// TIA Portal V20 export
TYPE "LConSMC_typeUnitConfiguration"
// Konfiguration der Einheiten / Configuration of the units
// stored: Access Published
   STRUCT
      metricUnits : Bool := TRUE;   // TRUE: Verwendung metrischer Einheiten [m] / [m/min] / [m/s^2] / [N] FALSE: Verwendung angloamerikanischer Einheiten [inch] / [ft/min] / [ft/s^2] / [Lbf] / TRUE: Use metric system [m] / [m/min] / [m/s^2] / [N] FALSE: Use angloamerican system [inch] / [ft/min] / [ft/s^2] / [Lbf]
      axisVelocityUnit : UDInt := 1083;   // Geschwindigkeitseinheit des Technologieobjektes (siehe TO.Units.VelocityUnit) !Nur notwendig wenn "getAxisConfigAtStart" = FALSE! / Velocity unit of TO (see TO.Units.VelocityUnit) !Only necessary if "getAxisConfigAtStart" = FALSE!
      axisTorqueUnit : UDInt := 1126;   // Drehmomenteinheit des Technologieobjektes (siehe TO.Units.TorqueUnit) !Nur notwendig wenn "getAxisConfigAtStart" = FALSE! / Torque unit of TO (see TO.Units.TorqueUnit) !Only necessary if "getAxisConfigAtStart" = FALSE!
   END_STRUCT;
END_TYPE
